FUNCTION_BLOCK FB_PlatoDivisor EXTENDS FB_Module
VAR_INPUT
	//tm			: REFERENCE TO FB_Timelimits;
	//tm			: FB_Timelimits;
	//TRET		: TIME := T#500MS;	(* Tiempo de actuación del retenedor del plato *)
	//TEMP	   	: TIME := T#2S   ;	(* Tiempo de recorrido del empujador del plato *)
END_VAR

VAR
	//tm: FB_Timelimits := (Speed:=10.0); //S_Timeouts;
	
	fbController: FB_PlatoDivisor_SFC;  // controlador para ejecución normal
	
	(* Sensores específicos *)
	d0 : dvSensor; //         AT %I*: BOOL; (* b0  (nombre=d0  c=I21 B=J1 b=29 módulo=EL1008 T=6  C=6 etiqueta=-B9,  input) Empujador del plato detrás *)
//    k1         AT %I*: BOOL; (* c1  (nombre=k1  c=I30 B=J1 b=15 módulo=EL1008 T=7  C=7 etiqueta=-B18, input) Empujador de tapa delante *)

	(* Actuadores específicos *)
    D_1       : dvActuator;// AT %Q*: BOOL; (* bEMP (nombre=D+  c=Q20 B=J2  b=05 módulo=EL2008 T=8 C=8 etiqueta=-Y6,  output) Empujador del plato avanza *)
    E_1       : dvActuator;// AT %Q*: BOOL; (* bRET (nombre=E+  c=Q21 B=J2  b=02 módulo=EL2008 T=8 C=8 etiqueta=-Y7,  output) Retenedor del plato retrocede *)

END_VAR

METHOD InitialConditions : BOOL
VAR_INPUT
END_VAR
InitialConditions := TRUE; // InitialConditions := d0;
END_METHOD

METHOD ModuleControlFlow : BOOL
//tm.UpdateSpeed(NewSpeed:= 0.01);
d0.ProcessCycle(gm.ModeActual, sfcValue=>fbController.d0);
IC := InitialConditions();
fbController(
	tm := tm, IC:=IC, Execute:=Execute, Ack:=Ack, Ready=>Ready, Done=>Done);
D_1.ProcessCycle(gm.ModeActual, sfcValue:=fbController.D_1);
E_1.ProcessCycle(gm.ModeActual, sfcValue:=fbController.E_1);
END_METHOD

END_FUNCTION_BLOCK

(* stored: Version 1.1.0.1, ProductVersion 3.1.4024.11
   POU FB_PlatoDivisor: Id {c71a4a01-3eb1-443b-a07e-accb57d2980d}, SpecialFunc None
   Method InitialConditions: Id {6c6766f3-90b7-4c0e-9ccf-d7be04fb6a0f}
   Method ModuleControlFlow: Id {a7156aed-454d-425e-80f1-664f90d71526} *)
